# EPICS substitutions: softIOC/halflinac/db/halflinac.substitutions
file db/quad.template {
  pattern {QUAD}
  { "QL01" }
  { "QL02" }
  { "QL03" }
  { "QL04" }
  { "QL05" }
  { "QL06" }
  { "QL07" }
  { "QL08" }
  { "QL09" }
  { "QL10" }
  { "QL11" }
  { "QL12" }
  { "QL13" }
  { "QL14" }
  { "QL15" }
  { "QL16" }
  { "QL17" }
  { "QL18" }
  { "QL19" }
  { "QL20" }
  { "QL21" }
  { "QL22" }
  { "QL23" }
  { "QL24" }
  { "QL25" }
  { "QL26" }
  { "QL27" }
  { "QT01" }
  { "QT02" }
  { "QT03" }
  { "QT04" }
  { "QHL1" }
  { "QHL2" }
  { "QHL3" }
  { "QHL4" }
  { "QT13" }
  { "QT14" }
  { "QT15" }
  { "QT16" }
  { "QTR1" }
  { "QT18" }
  { "QT19" }
  { "QT20" }
  { "QT21" }
  { "QT22" }
  { "QT23" }
  { "QT24" }
  { "QT25" }
  { "QT26" }
  { "QT27" }
  { "QT28" }
  { "QT29" }
  { "QT30" }
  { "QT31" }
  { "QT32" }
  { "QT33" }
  { "QT34" }
  { "QT35" }
  { "QT36" }
}
file db/bend.template {
  pattern {BEND}
  { "BH01" }
  { "BH02" }
  { "BH03" }
  { "BH04" }
  { "BV01" }
  { "BV02" }
  { "SEP2" }
  { "SEP1" }
}
file db/bpm.template {
  pattern {BPM}
  { "BPM01" }
  { "BPM02" }
  { "BPM03" }
  { "BPM04" }
  { "BPM05" }
  { "BPM06" }
  { "BPM07" }
  { "BPM08" }
  { "BPM09" }
  { "BPM10" }
  { "BPM11" }
  { "BPM12" }
  { "BPM13" }
  { "BPM14" }
  { "BPM15" }
  { "BPM16" }
  { "BPM17" }
  { "BPM18" }
  { "BPM19" }
  { "BPM20" }
  { "BPM21" }
  { "BPM22" }
  { "BPM23" }
  { "BPM24" }
  { "BPM25" }
  { "BPM26" }
  { "BPM27" }
  { "BPM28" }
  { "BPM29" }
  { "BPM30" }
  { "BPM31" }
  { "BPM32" }
  { "BPM33" }
  { "BPM34" }
  { "BPM35" }
  { "BPM36" }
  { "BPM37" }
  { "BPM38" }
  { "BPM39" }
  { "BPM40" }
  { "BPM41" }
  { "BPM42" }
  { "BPM43" }
}
file db/flag.template {
  pattern {FLAG}
  { "W00" }
  { "PRF02S" }
  { "FODO00" }
  { "PRF02" }
  { "PRF03" }
  { "PRF04" }
  { "FODO02" }
  { "FODO01" }
  { "PRF05" }
  { "FODO03" }
  { "FODO04" }
  { "PRF06" }
  { "PRF07" }
  { "PRF08" }
  { "PRF09" }
  { "FODO05" }
  { "PRF10" }
  { "WB1" }
  { "PRF11" }
  { "W01" }
  { "PRF12" }
  { "WB2" }
  { "PRF13" }
  { "PRF14" }
  { "WSEP1" }
}
file db/corr.template {
  pattern {COR}
  { "XC03" }
  { "XC04" }
  { "XC05" }
  { "XC06" }
  { "XC07" }
  { "XC08" }
  { "XC09" }
  { "XC10" }
  { "XC11" }
  { "XC12" }
  { "XC13" }
  { "XC14" }
  { "XC15" }
  { "XC16" }
  { "XC17" }
  { "XC18" }
  { "XC19" }
  { "XC20" }
  { "XC21" }
  { "XC22" }
  { "XC23" }
  { "XC24" }
  { "XC25" }
  { "XC26" }
  { "XC27" }
  { "XC28" }
  { "XC29" }
  { "XC30" }
  { "XC31" }
  { "XC32" }
  { "XC33" }
  { "XC34" }
  { "XC35" }
  { "XC36" }
  { "XC37" }
  { "XC38" }
  { "XC39" }
  { "XC40" }
  { "XC41" }
  { "XC42" }
  { "XC43" }
  { "YC03" }
  { "YC04" }
  { "YC05" }
  { "YC06" }
  { "YC07" }
  { "YC08" }
  { "YC09" }
  { "YC10" }
  { "YC11" }
  { "YC12" }
  { "YC13" }
  { "YC14" }
  { "YC15" }
  { "YC16" }
  { "YC17" }
  { "YC18" }
  { "YC19" }
  { "YC20" }
  { "YC21" }
  { "YC22" }
  { "YC23" }
  { "YC24" }
  { "YC25" }
  { "YC26" }
  { "YC27" }
  { "YC28" }
  { "YC29" }
  { "YC30" }
  { "YC31" }
  { "YC32" }
  { "YC33" }
  { "YC34" }
  { "YC35" }
  { "YC36" }
  { "YC37" }
  { "YC38" }
  { "YC39" }
  { "YC40" }
  { "YC41" }
  { "YC42" }
  { "YC43" }
}
